// TwinCAT 3 PLC project PLC1
// ProgramVersion: 3.1.4023.0
// libraries:
//   Tc2_MC2, * (Beckhoff Automation GmbH)
//   Tc2_Standard, * (Beckhoff Automation GmbH)
//   Tc2_System, * (Beckhoff Automation GmbH)
//   Tc3_Module, * (Beckhoff Automation GmbH)
//   XBoxControllerUtilities, * (Beckhoff Community)
// project tree:
//   / PlcTask.TcTTO
//   POUs/ MAIN.TcPOU
// real-time tasks:
//   TASK PlcTask: cycle T#10ms, priority 20, ADS port 350
// motion (NC):
//   TASK NC-Task 1 SAF: cycle T#2ms, priority 4, ADS port 501
//   TASK NC-Task 1 SVB: cycle T#10ms, priority 8, ADS port 511
//   AXIS Axis 1 (id 1)
//     OtherSettings: AllowMotionCmdToSlave=true
//     encoder EncType=1
//     drive DrvType=5
//       Analog: TorqueSetpointScale=10, ScaleFactorActTorque=0.1
//     controller CtrType=1
//       CtrPara: PriorControlFactor=1
//         Observer: BandWidth=20
//   AXIS Axis 2 (id 2)
//   AXIS Axis 3 (id 3)
// variable links:
//   PLC1 Instance <-> NC-Task 1 SAF/Axes/Axis 1
//     PlcTask Inputs/MAIN.Axis[1].NcToPlc <-> Outputs/ToPlc
//     PlcTask Outputs/MAIN.Axis[1].PlcToNc <-> Inputs/FromPlc
//   PLC1 Instance <-> NC-Task 1 SAF/Axes/Axis 2
//     PlcTask Inputs/MAIN.Axis[2].NcToPlc <-> Outputs/ToPlc
//     PlcTask Outputs/MAIN.Axis[2].PlcToNc <-> Inputs/FromPlc
//   PLC1 Instance <-> NC-Task 1 SAF/Axes/Axis 3
//     PlcTask Inputs/MAIN.Axis[3].NcToPlc <-> Outputs/ToPlc
//     PlcTask Outputs/MAIN.Axis[3].PlcToNc <-> Inputs/FromPlc

CONFIGURATION PLC1
    RESOURCE PLC ON TwinCAT3
        TASK PlcTask(INTERVAL := T#10ms, PRIORITY := 20);
        PROGRAM MAIN WITH PlcTask : MAIN;
    END_RESOURCE
END_CONFIGURATION

// ---- POUs/MAIN.TcPOU
PROGRAM MAIN
VAR
	XBoxController1 : FB_XBox_Controller('',1);	
	XBoxController2 : FB_XBox_Controller('',2);	
	JoystickJogger 	: FB_XBox_Dual_Directional_Joystick_NC;
	DualTrigger		: FB_XBox_Dual_Trigger_NC;
	
	Axis : ARRAY[1..3] OF AXIS_REF;
	Power : ARRAY[1..3] OF MC_Power;
	
	JoystickOp: ST_XBox_Dual_Directional_Joystick_NC_Options;
	TriggerOp: ST_XBox_Trigger_NC_Options;
END_VAR

XBoxController1.Cycle();
XBoxController2.Cycle();

Power[1](Axis:= Axis[1], Enable:= TRUE, Enable_Positive:= TRUE, Enable_Negative:= TRUE, Override:= 100);
Power[2](Axis:= Axis[2], Enable:= TRUE, Enable_Positive:= TRUE, Enable_Negative:= TRUE, Override:= 100);
Power[3](Axis:= Axis[3], Enable:= TRUE, Enable_Positive:= TRUE, Enable_Negative:= TRUE, Override:= 100);


JoystickJogger.Jog(bEnable := 	Power[1].Status AND Power[2].Status, 
								stJoystick := XBoxController1.P_Left_Joystick,
								X_Axis := Axis[1], Y_Axis := Axis[2],
								stOptions :=  JoystickOp);

DualTrigger.Jog(
				bEnable:= Power[3].Status, 
				fLeft_Trigger:= XBoxController2.P_Left_Trigger, 
				fRight_Trigger:= XBoxController2.P_Right_Trigger, 
				Axis:= Axis[3], 
				stOptions:= TriggerOp);

END_PROGRAM
